// TIA Portal V17 export
// export: Created 2024-06-16T17:47:25.6348883Z, ExportSetting WithDefaults, DisplayName Totally Integrated Automation Portal, DisplayVersion V17, DisplayName TIA Portal Openness, DisplayVersion V17, DisplayName TIA Portal Version Control Interface, DisplayVersion V17, DisplayName STEP 7 Professional, DisplayVersion V17, DisplayName STEP 7 Safety, DisplayVersion V17, DisplayName WinCC Professional, DisplayVersion V17
FUNCTION "G7A_St1" : Void   // FC105, LAD
{ S7_Optimized_Access := 'TRUE' }
VERSION : 0.1
// stored: AutoNumber false, IsIECCheckEnabled false, SetENOAutomatically false, UDAEnableTagReadback false
BEGIN

REGION Network 1: G7 Auto --> Station 1 : Empilement
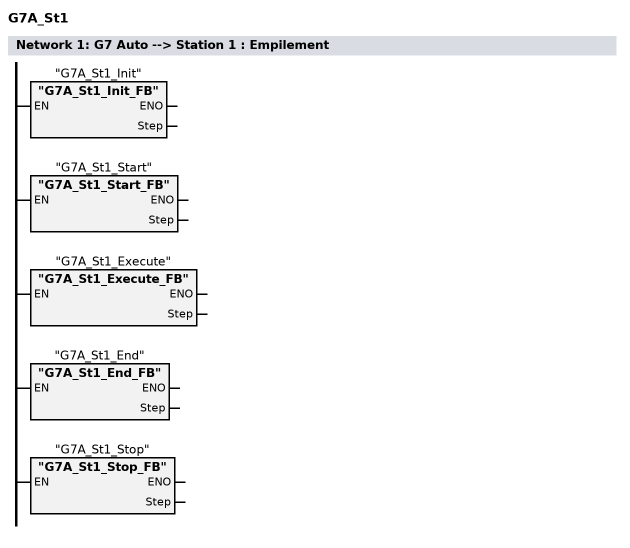
   RUNG wire#powerrail
      "G7A_St1_Init"("Step" =>)
   END_RUNG
   RUNG wire#powerrail
      "G7A_St1_Start"("Step" =>)
   END_RUNG
   RUNG wire#powerrail
      "G7A_St1_Execute"("Step" =>)
   END_RUNG
   RUNG wire#powerrail
      "G7A_St1_End"("Step" =>)
   END_RUNG
   RUNG wire#powerrail
      "G7A_St1_Stop"("Step" =>)
   END_RUNG
   // the same network as SCL:
   "G7A_St1_Init"();   // "G7A_St1_Init_FB"
   "G7A_St1_Start"();   // "G7A_St1_Start_FB"
   "G7A_St1_Execute"();   // "G7A_St1_Execute_FB"
   "G7A_St1_End"();   // "G7A_St1_End_FB"
   "G7A_St1_Stop"();   // "G7A_St1_Stop_FB"
END_REGION
END_FUNCTION
